Fanuc KAREL source: compact_preamble.KL

PROGRAM KB00005
%NOLOCKGROUP
VAR
P1 : STRING[80];P2 : STRING[80];P3 : STRING[80];P4:INTEGER;P5:INTEGER
BEGIN
P1='A'
P2='A'
P3='A'
P4=1
P5=1
ADD_DICT(P1,P2,P3,P4,P5)
END KB00005
